FUNCTION_BLOCK FB_MonetCabinetControl
VAR_INPUT
END_VAR
VAR_OUTPUT
	bCabinetOverTemp	: BOOL;	// cabinet temperature (BT1) is critical (>60°C); not wired to any stop/park action yet, see MONETcommon#21
END_VAR
VAR
	// AT%I*/AT%Q* below are mapped directly on this FB: only one instance per PLC is
	// supported, a second instance would collide on the same physical hardware.
	inKeyLocal			AT%I*: BOOL;	//DIN3 0.2
	inButtonStart		AT%I*: BOOL;	//DIN4 0.3
	inButtonStop		AT%I*: BOOL;	//DIN5 0.4
	inButtonReset		AT%I*: BOOL;	//DIN8 0.7
	inCabinetTemp		AT%I*: INT;		//BT1	
	inKeyClearBrakes	AT%I*: BOOL;	//DIN15 1.6
	outLampPower		AT%Q*: BOOL;	//DOUT1 0.0
	outLampManual		AT%Q*: BOOL;	//DOUT2 0.1
	outLampError		AT%Q*: BOOL;	//DOUT3 0.2	
	cabinetTemp				: REAL;
	tempWarning				: SR;
	tempCritical			: SR;
	tempEvent				: FB_EventLog;
	tempCriticalEvent		: FB_EventLog;
	blinkErrorLamp			: FB_BLINK;
	blinkPowerLamp			: FB_BLINK;
	commTimer 				: TON := (PT:=T#5S);
	fbComm					: I_Comm;
END_VAR

// check temperature
cabinetTemp := INT_TO_REAL(inCabinetTemp) / 10.0;
tempWarning(SET1 := cabinetTemp > 50.0, RESET := cabinetTemp < 40.0);
tempCritical(SET1 := cabinetTemp > 60.0, RESET := cabinetTemp < 50.0);
bCabinetOverTemp := tempCritical.Q1;

// blinking lights
blinkErrorLamp(Q => outLampError);
blinkPowerLamp(Q => outLampPower);

// telemetry
commTimer(IN:=TRUE);
IF commTimer.Q THEN
	commTimer(IN:=FALSE);
	fbComm.Publish('electronics', 'base', 'MainCabinetTemperature', LREAL_TO_FMTSTR(cabinetTemp, 2, TRUE));
END_IF

// events
tempEvent(	
	Trigger 		:= tempWarning.Q1, 
	Level 			:= ADSLOG_MSGTYPE_WARN,
	FormatString 	:= 'Main cabinet temperature warning:	%s',
	OnMessage 		:= LREAL_TO_FMTSTR(cabinetTemp, 1, TRUE),
	comm			:= fbComm);
tempCriticalEvent(	
	Trigger 		:= tempCritical.Q1, 
	Level 			:= ADSLOG_MSGTYPE_ERROR,
	FormatString 	:= 'Main cabinet temperature is critical:	%s!',
	OnMessage 		:= LREAL_TO_FMTSTR(cabinetTemp, 1, TRUE),
	comm			:= fbComm);

// deprecated: kept for existing callers (MONETN, MONETS MAIN), use AreBrakesCleared instead
METHOD PUBLIC AreBreakesCleared : BOOL
VAR_INPUT
END_VAR
AreBreakesCleared := THIS^.AreBrakesCleared();
END_METHOD

METHOD PUBLIC AreBrakesCleared : BOOL
VAR_INPUT
END_VAR
AreBrakesCleared := inKeyClearBrakes;
END_METHOD

//FB_Init is always available implicitly and it is used primarily for initialization.
//The return value is not evaluated. For a specific influence, you can also declare the
//methods explicitly and provide additional code there with the standard initialization
//code. You can evaluate the return value.
METHOD FB_Init: BOOL
VAR_INPUT
    bInitRetains	: BOOL; // TRUE: the retain variables are initialized (reset warm / reset cold)
    bInCopyCode		: BOOL;  // TRUE: the instance will be copied to the copy code afterward (online change)
	comm			: I_Comm;	   
END_VAR
THIS^.fbComm := comm;
END_METHOD

METHOD PUBLIC IsResetPushed : BOOL
VAR_INPUT
END_VAR
IsResetPushed := inButtonReset;
END_METHOD

METHOD PUBLIC IsStartPushed : BOOL
VAR_INPUT
END_VAR
IsStartPushed := inButtonStart;
END_METHOD

METHOD PUBLIC IsStopPushed : BOOL
VAR_INPUT
END_VAR
IsStopPushed := NOT inButtonStop;
END_METHOD

PROPERTY KeyLocal : BOOL
GET
KeyLocal := inKeyLocal;
END_GET
END_PROPERTY

METHOD PUBLIC SetBlinkError : BOOL
VAR_INPUT
	mode	: E_Blink;
END_VAR
blinkErrorLamp.blink := mode;
END_METHOD

METHOD PUBLIC SetBlinkPower : BOOL
VAR_INPUT
	mode	: E_Blink;
END_VAR
blinkPowerLamp.blink := mode;
END_METHOD

METHOD PUBLIC SetManualLamp : BOOL
VAR_INPUT
	enable	: BOOL;
END_VAR
outLampManual := enable;
END_METHOD

END_FUNCTION_BLOCK

(* stored: Version 1.1.0.1, ProductVersion 3.1.4024.15
   POU FB_MonetCabinetControl: Id {82301626-c59a-4d6c-ac78-2e8e2d6a8e41}, SpecialFunc None
   Method AreBreakesCleared: Id {febea358-d684-4605-9606-4cfb2e03d90b}
   Method AreBrakesCleared: Id {f1e9f4c4-2b3a-4a1e-9a4f-8f7e8f1c9d2a}
   Method FB_Init: Id {7d550def-2f64-47d1-ac2f-11dc091e5629}
   Method IsResetPushed: Id {c5f0543d-d2ee-4085-9cc6-f6a37ba59d95}
   Method IsStartPushed: Id {1ca9b4ce-3543-45dd-a0d5-ec2fcef43780}
   Method IsStopPushed: Id {2e5a1388-2bbb-4716-8012-08858212fbd5}
   Property KeyLocal: Id {ad8e8c92-5a56-4bc4-94dd-dcc3a456a9f1}
   Get Get: Id {8be1cdac-bba1-4a4a-bac4-cea38f645137}
   Method SetBlinkError: Id {f01ddc4d-dc53-44dc-b62c-672aa08804ee}
   Method SetBlinkPower: Id {0c127d75-c801-44ba-a87e-6f0d74dad2e5}
   Method SetManualLamp: Id {bad59df7-0faf-454c-875d-08335ce28698} *)
